// TIA Portal V16 export
// export: Created 2024-06-18T17:34:29.501273Z, ExportSetting WithDefaults, DisplayName Totally Integrated Automation Portal, DisplayVersion V16, DisplayName TIA Portal Version Control Interface, DisplayVersion V16, DisplayName TIA Portal Openness, DisplayVersion V16, DisplayName STEP 7 Professional, DisplayVersion V16, DisplayName STEP 7 Safety, DisplayVersion V16, DisplayName WinCC Advanced, DisplayVersion V16
TYPE "Axis.RB_Memórias_Internas"
TITLE = RB_Memórias Internas
// Essa Memorias são escritas pelo software DENTRO do bloco do robô
// stored: IsFailsafeCompliant false
   STRUCT
      RB_F_RS : Bool;   // RB - Memoria Robo Start
      RB_Prog_OK : Bool;   // RB - Programa ok
      RB_Aux_RST_P_OK : Bool;   // RB - Auxiliar Reset Programa OK
      RB_Pulso_RST_P_OK : Bool;   // RB - Pulso Reset Programa OK
      SA_G : Bool;   // RB - SEGURANÇA GERAL
      SA_A : Bool;   // RB - SEGURANÇA COM ROBO EM AUTOMÁTICO
      SA_P : Bool;   // RB - SEGURANÇA PARA CHAMADA PROGRAMA ROBO
      Sts_Automatico : Bool;   // RB - Status Robô em Automático sem Falha
      Sts_Manual : Bool;   // RB - Status Robô em Manual
      Sts_Falha : Bool;   // RB - Status Robô em Falha
      "Nenhuma Chamada Ativa" : Bool;   // RB - Resolutivo de Chamada de Programa / Nenhuma chamada de programa ativa
      RB_Mem_Prog_RB_Enviado : Int;   // RB - Numero de Programa Enviado pelo PLC para Robô / Número de programa ENVIADO ao Robo
      RB_Mem_Prog_RB_Recebido : Int;   // RB - Numero de Programa Enviado pelo Robô para PLC / Número de programa RECEBIDO do Robo
   END_STRUCT;
END_TYPE
